# EPICS substitutions: LS336/LS336-IOC-01App/Db/LS336.substitutions
file $(LAKESHORE336)/db/lakeshore336.template
{
pattern {P, PORT, ADDR, TEMPSCAN, SCAN}
	{\$(P):LS01, L0, 0, 1, 5}
}
